FUNCTION_BLOCK FB_TcBSD_Backup
VAR_INPUT
END_VAR
VAR_OUTPUT
END_VAR
VAR
//SMTP Sendmail
	fbTcBackup:NT_StartProcess;			//SytemBackup
	
//Mail Sendstring
	sCommand:STRING(512);				//Command
	
//Execute
	bProcessExecute:BOOL;				//Process Execute
	bProcessActive:BOOL;				//Process Active
	bProcessBusy:BOOL;					//Process Busy
	bProcessError:BOOL;					//Process Error
	
//Bacup Parameter
	sBackupDisk:STRING;					//Backup Disk
	sBackupName:STRING;					//Backup Name
	sBackupFolder:STRING;				//backup Folder
	
//Status & Helper
	tonExecuteReset: TON;				//Timer Execute Reset
	
END_VAR

PROPERTY BackupDisk : STRING
SET
sBackupDisk:=BackupDisk;
END_SET
END_PROPERTY

PROPERTY BackupFolder : STRING
SET
sBackupFolder:=BackupFolder;
END_SET
END_PROPERTY

PROPERTY BackupName : STRING
SET
sBackupName:=BackupName;
END_SET
END_PROPERTY

METHOD BuildCommand : INT
VAR_INPUT
END_VAR
//Build Commans
sCommand:= '"TcBackup.sh --disk ';
sCommand:=CONCAT(sCommand, sBackupDisk);
sCommand:=CONCAT(sCommand, ' > ');
sCommand:=CONCAT(sCommand, sBackupFolder);
sCommand:=CONCAT(sCommand, '/');
sCommand:=CONCAT(sCommand, sBackupName);
sCommand:=CONCAT(sCommand, '.tcbkp00');
sCommand:=CONCAT(sCommand, '"');
END_METHOD

METHOD Cyclic : INT
VAR_INPUT
END_VAR
(*

--Call Cyclic

*)

BuildCommand();

//Send Mail
fbTcBackup(
	NETID:= '', 
	PATHSTR:='/bin/sh -c' , 
	DIRNAME:='/bin' , 
	COMNDLINE:=sCommand , 
	START:=bProcessActive, 
	TMOUT:= , 
	BUSY=> , 
	ERR=> , 
	ERRID=> );

//Send Execute Reset		
tonExecuteReset(IN:=bProcessExecute=FALSE AND bProcessActive=TRUE , PT:=T#5S);
IF tonExecuteReset.Q THEN
	bProcessActive:=FALSE;
END_IF
bProcessExecute:=FALSE;

//Status Signals
bProcessBusy:=bProcessActive;
IF bProcessActive AND fbTcBackup.ERR THEN
	bProcessError:=TRUE;
END_IF
END_METHOD

METHOD Execute : INT
VAR_INPUT
END_VAR
//Execute

//Build Build Command
BuildCommand();

//Flag Securtiy
if bProcessExecute=false then
	bProcessActive:=TRUE;
	bProcessError:=FALSE;
END_IF
bProcessExecute:=TRUE;
END_METHOD

END_FUNCTION_BLOCK

(* stored: Version 1.1.0.1, ProductVersion 3.1.4024.12
   POU FB_TcBSD_Backup: Id {a42133b4-5218-4b11-84a7-7021528c6850}, SpecialFunc None
   Property BackupDisk: Id {85993fb2-d085-4c48-a11f-8bec90b32b56}
   Set Set: Id {2435e079-ea52-4947-a5ea-e86e8f161f25}
   Property BackupFolder: Id {db37a17d-f742-4081-bce6-afb74dbfc25e}
   Set Set: Id {6bdcb3a1-7831-42d3-9fd6-950ab6d6cda0}
   Property BackupName: Id {ef5f9fd3-1283-4080-b1dd-9e71a7e5e190}
   Set Set: Id {5a6e5f18-096c-4a70-804b-3dc0316265b7}
   Method BuildCommand: Id {9284c032-7138-4c10-b52e-66008292f816}
   Method Cyclic: Id {b45cbff1-d2d2-496d-ae8c-f1b35ca7a815}
   Method Execute: Id {e3fe95f1-6a65-40a0-a1ad-8ff80552c941} *)
